{attribute 'linkalways'} 
{attribute 'no_explicit_call' := 'This FB is a CLASS and must be accessed using methods or properties'}
{attribute 'enable_dynamic_creation'}
FUNCTION_BLOCK FINAL XOR_DWORD EXTENDS Node
VAR
	in1 : _DWORD(0);
	in2 : _DWORD(0);
	out : _DWORD(0);
END_VAR

METHOD PUBLIC Clone : I_Node
VAR
	pNode : POINTER TO XOR_DWORD;
END_VAR
pNode := __NEW(XOR_DWORD);
Clone := pNode^;
END_METHOD

METHOD FB_init : BOOL
VAR_INPUT
	bInitRetains : BOOL; // if TRUE, the retain variables are initialized (warm start / cold start)
	bInCopyCode : BOOL;  // if TRUE, the instance afterwards gets moved into the copy code (online change)
END_VAR
AddInput('in1',THIS^.in1);
AddInput('in2',THIS^.in2);
AddOutput('out', THIS^.out);
END_METHOD

METHOD PROTECTED OnExecute
VAR
END_VAR
out.Value := in1.Value XOR in2.Value;
END_METHOD

END_FUNCTION_BLOCK

(* stored: Version 1.1.0.1, ProductVersion 3.1.4024.15
   POU XOR_DWORD: Id {9ee0df70-5798-4687-b338-280c346a4d64}, SpecialFunc None
   Folder Constructor: Id {d99fa16d-4279-4477-a818-aadf91db0b47}
   Method Clone: Id {7094b97c-0450-4517-9c84-57b5ae10be27}
   Method FB_init: Id {da163aab-c331-4570-9bf8-56f5296755b3}
   Method OnExecute: Id {3feec2b2-dc6f-404f-ae56-ab684816e000} *)
